(* IEC 61131-3 sources: RAG_PLC/data/result/test/066, 2 files *)

(* ---- wrapped.st ---- *)
(* =========================================================
   Generated by PLC-Eval Benchmark Wrapper
   ========================================================= *)

FUNCTION_BLOCK LLM_Wrapper_FB
VAR_INPUT
	A : oscat_vector_3;
END_VAR

VAR_OUTPUT
	V3_XANG : REAL;
END_VAR

VAR
	la : REAL;
	V3_ABS : V3_ABS;
END_VAR

V3_ABS(A:=A);
la := V3_ABS.V3_ABS;

IF la > 0.0 THEN
	V3_XANG := ACOS(A.X / la);
ELSE
	V3_XANG := 0.0;
END_IF;
END_FUNCTION_BLOCK

PROGRAM Auto_Proxy_Prg
  VAR
    instance : LLM_Wrapper_FB;
  END_VAR

  instance();
END_PROGRAM

CONFIGURATION Config0
  RESOURCE Res0 ON PLC
    TASK TaskMain(INTERVAL := T#20ms, PRIORITY := 0);
    PROGRAM Inst0 WITH TaskMain : Auto_Proxy_Prg;
  END_RESOURCE
END_CONFIGURATION

(* ---- raw_code.st ---- *)
VAR_INPUT
	A : oscat_vector_3;
END_VAR

VAR_OUTPUT
	V3_XANG : REAL;
END_VAR

VAR
	la : REAL;
	V3_ABS : V3_ABS;
END_VAR

V3_ABS(A:=A);
la := V3_ABS.V3_ABS;

IF la > 0.0 THEN
	V3_XANG := ACOS(A.X / la);
ELSE
	V3_XANG := 0.0;
END_IF;
